Yaskawa INFORM job: TABLE_TEST.JBI

/JOB
//NAME TABLE_TEST
//POS
///NPOS 1,0,1,0,0,0
///TOOL 0
///POSTYPE BASE
///RECTAN
///RCONF 1,0,0,0,0,0,0,0,0,0,0,0,0,0,0,0,0,0,0,0,0,0,0,0
C00000=2270.9747,-236.3144,-436.5992,0.0000,0.0000,0.0000
EC00000=0.0000,0.0000,0.0000,0.000000,0.0000,180.0000
//INST
///DATE 2023/01/12 15:59
///ATTR SC,RW
///GROUP1 RB1,ST1
NOP
MOVJ C00000 EC00000 VJ=0.78
END
